# EPICS substitutions: rogueApp/Db/Integrators.substitutions
# Integrators.substitutions

file liDevRogue.template
{
	{
		NAME	= "Integrators:AdcIntegral0",
		PATH	= "Top.Integrators.AdcIntegral[0]"
		PYPV	= "AdcIntegral0"
		DESC	= "Integration of A/D value"
		SCAN	= "I/O Intr"
		PRIO	= "HIGH"
		TSE		= "-2"
		R       = ":Fast\$(R)"
	}
	{
		NAME	= "Integrators:AdcIntegral1",
		PATH	= "Top.Integrators.AdcIntegral[1]"
		PYPV	= "AdcIntegral1"
		DESC	= "Integration of A/D value"
		SCAN	= "I/O Intr"
		PRIO	= "HIGH"
		TSE		= "-2"
		R       = ":Fast\$(R)"
	}
	{
		NAME	= "Integrators:AdcIntegral2",
		PATH	= "Top.Integrators.AdcIntegral[2]"
		PYPV	= "AdcIntegral2"
		DESC	= "Integration of A/D value"
		SCAN	= "I/O Intr"
		PRIO	= "HIGH"
		TSE		= "-2"
		R       = ":Fast\$(R)"
	}
	{
		NAME	= "Integrators:AdcIntegral3",
		PATH	= "Top.Integrators.AdcIntegral[3]"
		PYPV	= "AdcIntegral3"
		DESC	= "Integration of A/D value"
		SCAN	= "I/O Intr"
		PRIO	= "HIGH"
		TSE		= "-2"
		R       = ":Fast\$(R)"
	}
	{
		NAME	= "Integrators:AdcIntegral4",
		PATH	= "Top.Integrators.AdcIntegral[4]"
		PYPV	= "AdcIntegral4"
		DESC	= "Integration of A/D value"
		SCAN	= "I/O Intr"
		PRIO	= "HIGH"
		TSE		= "-2"
		R       = ":Fast\$(R)"
	}
	{
		NAME	= "Integrators:AdcIntegral5",
		PATH	= "Top.Integrators.AdcIntegral[5]"
		PYPV	= "AdcIntegral5"
		DESC	= "Integration of A/D value"
		SCAN	= "I/O Intr"
		PRIO	= "HIGH"
		TSE		= "-2"
		R       = ":Fast\$(R)"
	}
	{
		NAME	= "Integrators:AdcIntegral6",
		PATH	= "Top.Integrators.AdcIntegral[6]"
		PYPV	= "AdcIntegral6"
		DESC	= "Integration of A/D value"
		SCAN	= "I/O Intr"
		PRIO	= "HIGH"
		TSE		= "-2"
		R       = ":Fast\$(R)"
	}
	{
		NAME	= "Integrators:AdcIntegral7",
		PATH	= "Top.Integrators.AdcIntegral[7]"
		PYPV	= "AdcIntegral7"
		DESC	= "Integration of A/D value"
		SCAN	= "I/O Intr"
		PRIO	= "HIGH"
		TSE		= "-2"
		R       = ":Fast\$(R)"
	}
	{
		NAME	= "Integrators:AdcIntegral0",
		PATH	= "Top.Integrators.AdcIntegral[0]"
		PYPV	= "Top:Integrators:AdcIntegral[0]"
		DESC	= "Integration of A/D value"
		SCAN	= "\$(SCAN=.1 second)"
	}
	{
		NAME	= "Integrators:AdcIntegral1",
		PATH	= "Top.Integrators.AdcIntegral[1]"
		PYPV	= "Top:Integrators:AdcIntegral[1]"
		DESC	= "Integration of A/D value"
		SCAN	= "\$(SCAN=.1 second)"
	}
	{
		NAME	= "Integrators:AdcIntegral2",
		PATH	= "Top.Integrators.AdcIntegral[2]"
		PYPV	= "Top:Integrators:AdcIntegral[2]"
		DESC	= "Integration of A/D value"
		SCAN	= "\$(SCAN=.1 second)"
	}
	{
		NAME	= "Integrators:AdcIntegral3",
		PATH	= "Top.Integrators.AdcIntegral[3]"
		PYPV	= "Top:Integrators:AdcIntegral[3]"
		DESC	= "Integration of A/D value"
		SCAN	= "\$(SCAN=.1 second)"
	}
	{
		NAME	= "Integrators:AdcIntegral4",
		PATH	= "Top.Integrators.AdcIntegral[4]"
		PYPV	= "Top:Integrators:AdcIntegral[4]"
		DESC	= "Integration of A/D value"
		SCAN	= "\$(SCAN=.1 second)"
	}
	{
		NAME	= "Integrators:AdcIntegral5",
		PATH	= "Top.Integrators.AdcIntegral[5]"
		PYPV	= "Top:Integrators:AdcIntegral[5]"
		DESC	= "Integration of A/D value"
		SCAN	= "\$(SCAN=.1 second)"
	}
	{
		NAME	= "Integrators:AdcIntegral6",
		PATH	= "Top.Integrators.AdcIntegral[6]"
		PYPV	= "Top:Integrators:AdcIntegral[6]"
		DESC	= "Integration of A/D value"
		SCAN	= "\$(SCAN=.1 second)"
	}
	{
		NAME	= "Integrators:AdcIntegral7",
		PATH	= "Top.Integrators.AdcIntegral[7]"
		PYPV	= "Top:Integrators:AdcIntegral[7]"
		DESC	= "Integration of A/D value"
		SCAN	= "\$(SCAN=.1 second)"
	}
}

file boolDevRogue.template
{
	{
		NAME	= "Integrators:CntRst",
		PATH	= "Top.Integrators.CntRst"
		PYPV	= "Top:Integrators:CntRst"
		PINI	= ""
		SCAN	= "\$(SCAN=1 second)"
	}
	{
		NAME	= "Integrators:QuadrantSel",
		PATH	= "Top.Integrators.QuadrantSel"
		PYPV	= "Top:Integrators:QuadrantSel"
		DESC	= "Ch0-3 vs Ch4-7 for float equations"
		PINI	= "YES"
		SCAN	= ""
		ZNAM	= "Ch0-3"
		ONAM	= "Ch4-7"
	}
}

file liDevRogue.template
{
	{
		NAME	= "Integrators:Baseline0",
		PATH	= "Top.Integrators.Baseline[0]"
		PYPV	= "Top:Integrators:Baseline[0]"
		DESC	= "Baseline for integration"
		SCAN	= "\$(SCAN=1 second)"
		EGU		= "Pwr2"
	}
	{
		NAME	= "Integrators:Baseline1",
		PATH	= "Top.Integrators.Baseline[1]"
		PYPV	= "Top:Integrators:Baseline[1]"
		DESC	= "Baseline for integration"
		SCAN	= "\$(SCAN=1 second)"
		EGU		= "Pwr2"
	}
	{
		NAME	= "Integrators:Baseline2",
		PATH	= "Top.Integrators.Baseline[2]"
		PYPV	= "Top:Integrators:Baseline[2]"
		DESC	= "Baseline for integration"
		SCAN	= "\$(SCAN=1 second)"
		EGU		= "Pwr2"
	}
	{
		NAME	= "Integrators:Baseline3",
		PATH	= "Top.Integrators.Baseline[3]"
		PYPV	= "Top:Integrators:Baseline[3]"
		DESC	= "Baseline for integration"
		SCAN	= "\$(SCAN=1 second)"
		EGU		= "Pwr2"
	}
	{
		NAME	= "Integrators:Baseline4",
		PATH	= "Top.Integrators.Baseline[4]"
		PYPV	= "Top:Integrators:Baseline[4]"
		DESC	= "Baseline for integration"
		SCAN	= "\$(SCAN=1 second)"
		EGU		= "Pwr2"
	}
	{
		NAME	= "Integrators:Baseline5",
		PATH	= "Top.Integrators.Baseline[5]"
		PYPV	= "Top:Integrators:Baseline[5]"
		DESC	= "Baseline for integration"
		SCAN	= "\$(SCAN=1 second)"
		EGU		= "Pwr2"
	}
	{
		NAME	= "Integrators:Baseline6",
		PATH	= "Top.Integrators.Baseline[6]"
		PYPV	= "Top:Integrators:Baseline[6]"
		DESC	= "Baseline for integration"
		SCAN	= "\$(SCAN=1 second)"
		EGU		= "Pwr2"
	}
	{
		NAME	= "Integrators:Baseline7",
		PATH	= "Top.Integrators.Baseline[7]"
		PYPV	= "Top:Integrators:Baseline[7]"
		DESC	= "Baseline for integration"
		SCAN	= "\$(SCAN=1 second)"
		EGU		= "Pwr2"
	}
	{
		NAME	= "Integrators:IntFifoPauseCnt",
		PATH	= "Top.Integrators.IntFifoPauseCnt"
		PYPV	= "Top:Integrators:IntFifoPauseCnt"
		PINI	= "YES"
		SCAN	= "\$(SCAN=1 second)"
	}
	{
		NAME	= "Integrators:ProcFifoPauseCnt",
		PATH	= "Top.Integrators.ProcFifoPauseCnt"
		PYPV	= "Top:Integrators:ProcFifoPauseCnt"
		SCAN	= "\$(SCAN=1 second)"
	}
}

file longDevRogue.template
{
    {
        NAME    = "Integrators:IntegralSigned",
        PATH    = "Top.Integrators.IntegralSigned"
        PYPV    = "Top:Integrators:IntegralSigned"
        DESC    = "Carry Integral sign"
        PINI    = "YES"
        SAVE    = "VAL"
        SCAN    = "\$(SCAN=1 second)"
    }
	{
		NAME	= "Integrators:BaselineSize",
		PATH	= "Top.Integrators.BaselineSize"
		PYPV	= "Top:Integrators:BaselineSize"
		DESC	= "Baseline sample size as power of 2"
		PINI	= "YES"
		DOL	= "7"
		SAVE	= "VAL"
		EGU	= "2^X"
		SCAN	= "\$(SCAN=1 second)"
	}
	{
		NAME	= "Integrators:CorrCoefficientRaw0",
		PATH	= "Top.Integrators.CorrCoefficientRaw[0]"
		PYPV	= "Top:Integrators:CorrCoefficientRaw[0]"
		DESC	= "Gain correction coefficient 0 in Float64"
		PINI	= "YES"
		SCAN	= ""
	}
	{
		NAME	= "Integrators:CorrCoefficientRaw1",
		PATH	= "Top.Integrators.CorrCoefficientRaw[1]"
		PYPV	= "Top:Integrators:CorrCoefficientRaw[1]"
		DESC	= "Gain correction coefficient 1 in Float64"
		PINI	= "YES"
		SCAN	= ""
	}
	{
		NAME	= "Integrators:CorrCoefficientRaw2",
		PATH	= "Top.Integrators.CorrCoefficientRaw[2]"
		PYPV	= "Top:Integrators:CorrCoefficientRaw[2]"
		DESC	= "Gain correction coefficient 2 in Float64"
		PINI	= "YES"
		SCAN	= ""
	}
	{
		NAME	= "Integrators:CorrCoefficientRaw3",
		PATH	= "Top.Integrators.CorrCoefficientRaw[3]"
		PYPV	= "Top:Integrators:CorrCoefficientRaw[3]"
		DESC	= "Gain correction coefficient 3 in Float64"
		PINI	= "YES"
		SCAN	= ""
	}
	{
		NAME	= "Integrators:IntFifoPauseThreshold",
		PATH	= "Top.Integrators.IntFifoPauseThreshold"
		PYPV	= "Top:Integrators:IntFifoPauseThreshold"
		PINI	= "YES"
		DOL	= "255"
		SCAN	= ""
	}
	{
		NAME	= "Integrators:IntegralSize",
		PATH	= "Top.Integrators.IntegralSize"
		PYPV	= "Top:Integrators:IntegralSize"
		DESC	= "Integral sample size as # samples"
		DOL	= "1"
		SAVE	= "VAL"
		PINI	= "YES"
		EGU	= "Samples"
		SCAN	= ""
		SCAN	= "\$(SCAN=1 second)"
	}
	{
		NAME	= "Integrators:ProcFifoPauseThreshold",
		PATH	= "Top.Integrators.ProcFifoPauseThreshold"
		PYPV	= "Top:Integrators:ProcFifoPauseThreshold"
		PINI	= "YES"
		DOL	= "255"
		SAVE	= "VAL"
		SCAN	= "\$(SCAN=1 second)"
	}
	{
		NAME	= "Integrators:TrigDelay",
		PATH	= "Top.Integrators.TrigDelay"
		PYPV	= "Top:Integrators:TrigDelay"
		DESC	= "Integrator start offset in samples"
		DOL	= "5"
		SAVE	= "VAL"
		PINI	= "YES"
		EGU	= "Samples"
		SCAN	= ""
		SCAN	= "\$(SCAN=1 second)"
	}
}

file int64InDevRogue.template
{
	{
		NAME	= "Integrators:IntensityRaw",
		PATH	= "Top.Integrators.IntensityRaw"
		PYPV	= "Top:Integrators:IntensityRaw"
		PINI	= "YES"
		SCAN	= "\$(SCAN=.1 second)"
	}
	{
		NAME	= "Integrators:PositionXRaw",
		PATH	= "Top.Integrators.PositionXRaw"
		PYPV	= "Top:Integrators:PositionXRaw"
		PINI	= "YES"
		SCAN	= "\$(SCAN=.1 second)"
	}
	{
		NAME	= "Integrators:PositionYRaw",
		PATH	= "Top.Integrators.PositionYRaw"
		PYPV	= "Top:Integrators:PositionYRaw"
		PINI	= "YES"
		SCAN	= "\$(SCAN=.1 second)"
	}
	{
		NAME	= "Integrators:TrigCnt",
		PATH	= "Top.Integrators.TrigCnt"
		PYPV	= "Top:Integrators:TrigCnt"
		PINI	= "YES"
		SCAN	= "\$(SCAN=1 second)"
	}
}
#       DESC    = "0         1         2         3         "
#       DESC    = "01234567890123 Max 40 char 7890123456789"
